// TIA Portal V20 export
DATA_BLOCK "BK33"   // DB236
// stored: MemoryReserve 100
   VAR
      "X10-1.ANODE MAIN P&P1-2 VACUUM ON" : Bool := FALSE;
      "X10-2.ANODE MAIN P&P1-2 VACUUM OFF" : Bool := FALSE;
      "X12-1.CATHODE MAIN P&P1-2 VACUUM ON" : Bool := FALSE;
      "X12-2.CATHODE MAIN P&P1-2 VACUUM OFF" : Bool := FALSE;
      "X14-1.ANODE MAIN P&P2-2 VACUUM ON" : Bool := FALSE;
      "X14-2.ANODE MAIN P&P2-2 VACUUM OFF" : Bool := FALSE;
      "X16-1.CATHODE MAIN P&P2-2 VACUUM ON" : Bool := FALSE;
      "X16-2.CATHODE MAIN P&P2-2 VACUUM OFF" : Bool := FALSE;
   END_VAR
BEGIN
END_DATA_BLOCK
